# EPICS autosave request: zmqApp/Db/ADZMQ_settings.req
$(P)$(R)TopicID
file "NDPluginBase_settings.req", P=$(P), R=$(R)
